// TIA Portal V20 export
TYPE "UDT_MTP_AnaServParam_Recipe"
   STRUCT
      V : Real;   // External parameter value variable; relevant, if StateAutAct is true and SrcExtAct is true
      VFbk { ExternalWritable := 'False'} : Real;   // Feedback value variable
      VSclMin { ExternalWritable := 'False'} : Real;   // value scale low limit
      VSclMax { ExternalWritable := 'False'} : Real := 100.0;   // value scale high limit
      VUnit { ExternalWritable := 'False'} : Int := 1998;   // value unit
      VMin { ExternalWritable := 'False'} : Real;   // value low limit
      VMax { ExternalWritable := 'False'} : Real := 100.0;   // value high limit
      V_1 : Real;
      VFbk_1 : Real;
      VSclMin_1 : Real;
      VSclMax_1 : Real;
      VUnit_1 : Real;
      VMin_1 : Real;
      VMax_1 : Real;
      V_2 : Real;
      VFbk_2 : Real;
      VSclMin_2 : Real;
      VSclMax_2 : Real;
      VUnit_2 : Real;
      VMin_2 : Real;
      VMax_2 : Real;
      V_3 : Real;
      VFbk_3 : Real;
      VSclMin_3 : Real;
      VSclMax_3 : Real;
      VUnit_3 : Real;
      VMin_3 : Real;
      VMax_3 : Real;
      V_4 : Real;
      VFbk_4 : Real;
      VSclMin_4 : Real;
      VSclMax_4 : Real;
      VUnit_4 : Real;
      VMin_4 : Real;
      VMax_4 : Real;
      V_5 : Real;
      VFbk_5 : Real;
      VSclMin_5 : Real;
      VSclMax_5 : Real;
      VUnit_5 : Real;
      VMin_5 : Real;
      VMax_5 : Real;
      V_6 : Real;
      VFbk_6 : Real;
      VSclMin_6 : Real;
      VSclMax_6 : Real;
      VUnit_6 : Real;
      VMin_6 : Real;
      VMax_6 : Real;
      V_7 : Real;
      VFbk_7 : Real;
      VSclMin_7 : Real;
      VSclMax_7 : Real;
      VUnit_7 : Real;
      VMin_7 : Real;
      VMax_7 : Real;
      V_8 : Real;
      VFbk_8 : Real;
      VSclMin_8 : Real;
      VSclMax_8 : Real;
      VUnit_8 : Real;
      VMin_8 : Real;
      VMax_8 : Real;
      V_9 : Real;
      VFbk_9 : Real;
      VSclMin_9 : Real;
      VSclMax_9 : Real;
      VUnit_9 : Real;
      VMin_9 : Real;
      VMax_9 : Real;
      V_10 : Real;
      VFbk_10 : Real;
      VSclMin_10 : Real;
      VSclMax_10 : Real;
      VUnit_10 : Real;
      VMin_10 : Real;
      VMax_10 : Real;
      V_11 : Real;
      VFbk_11 : Real;
      VSclMin_11 : Real;
      VSclMax_11 : Real;
      VUnit_11 : Real;
      VMin_11 : Real;
      VMax_11 : Real;
      V_12 : Real;
      VFbk_12 : Real;
      VSclMin_12 : Real;
      VSclMax_12 : Real;
      VUnit_12 : Real;
      VMin_12 : Real;
      VMax_12 : Real;
      V_13 : Real;
      VFbk_13 : Real;
      VSclMin_13 : Real;
      VSclMax_13 : Real;
      VUnit_13 : Real;
      VMin_13 : Real;
      VMax_13 : Real;
      V_14 : Real;
      VFbk_14 : Real;
      VSclMin_14 : Real;
      VSclMax_14 : Real;
      VUnit_14 : Real;
      VMin_14 : Real;
      VMax_14 : Real;
      V_15 : Real;
      VFbk_15 : Real;
      VSclMin_15 : Real;
      VSclMax_15 : Real;
      VUnit_15 : Real;
      VMin_15 : Real;
      VMax_15 : Real;
      V_16 : Real;
      VFbk_16 : Real;
      VSclMin_16 : Real;
      VSclMax_16 : Real;
      VUnit_16 : Real;
      VMin_16 : Real;
      VMax_16 : Real;
      V_17 : Real;
      VFbk_17 : Real;
      VSclMin_17 : Real;
      VSclMax_17 : Real;
      VUnit_17 : Real;
      VMin_17 : Real;
      VMax_17 : Real;
      V_18 : Real;
      VFbk_18 : Real;
      VSclMin_18 : Real;
      VSclMax_18 : Real;
      VUnit_18 : Real;
      VMin_18 : Real;
      VMax_18 : Real;
      V_19 : Real;
      VFbk_19 : Real;
      VSclMin_19 : Real;
      VSclMax_19 : Real;
      VUnit_19 : Real;
      VMin_19 : Real;
      VMax_19 : Real;
      V_20 : Real;
      VFbk_20 : Real;
      VSclMin_20 : Real;
      VSclMax_20 : Real;
      VUnit_20 : Real;
      VMin_20 : Real;
      VMax_20 : Real;
   END_STRUCT;
END_TYPE
